{attribute 'linkalways'} 
{attribute 'no_explicit_call' := 'This FB is a CLASS and must be accessed using methods or properties'}
{attribute 'enable_dynamic_creation'}
FUNCTION_BLOCK _ETcVnTemplateMatchMethod EXTENDS EnumDatatypeBase
VAR
	localData : ETcVnTemplateMatchMethod;
	activeData : REFERENCE TO ETcVnTemplateMatchMethod;
	enumBaseDatatype : _DINT(localData);
END_VAR

METHOD PRIVATE AddLocalEnumeration
VAR_INPUT
	Enumeration : T_MAXSTRING;
	Value : ETcVnTemplateMatchMethod;
END_VAR
AddEnumeration(Enumeration, Value);
END_METHOD

PROPERTY PUBLIC Address : PVOID
GET
Address := ADR(activeData);
END_GET
END_PROPERTY

METHOD PUBLIC ClearReference
VAR_INPUT
END_VAR
activeData REF= localData;
SetBaseDatatypeReference();
END_METHOD

METHOD PUBLIC Clone : I_Datatype
VAR
    pClone : POINTER TO _ETcVnTemplateMatchMethod;
END_VAR
pClone := __NEW(_ETcVnTemplateMatchMethod(InitialValue := Value));
Clone := pClone^;
END_METHOD

METHOD FB_init : BOOL
VAR_INPUT
	bInitRetains : BOOL; // if TRUE, the retain variables are initialized (warm start / cold start)
	bInCopyCode : BOOL;  // if TRUE, the instance afterwards gets moved into the copy code (online change)
	InitialValue : ETcVnTemplateMatchMethod;
END_VAR
localData := InitialValue;
AddBaseDatatype(enumBaseDatatype);
ClearReference();

AddLocalEnumeration('TCVN_TMM_SQDIFF', ETcVnTemplateMatchMethod.TCVN_TMM_SQDIFF);
AddLocalEnumeration('TCVN_TMM_SQDIFF_NORMED', ETcVnTemplateMatchMethod.TCVN_TMM_SQDIFF_NORMED);
AddLocalEnumeration('TCVN_TMM_CCORR', ETcVnTemplateMatchMethod.TCVN_TMM_CCORR);
AddLocalEnumeration('TCVN_TMM_CCORR_NORMED', ETcVnTemplateMatchMethod.TCVN_TMM_CCORR_NORMED);
AddLocalEnumeration('TCVN_TMM_CCOEFF', ETcVnTemplateMatchMethod.TCVN_TMM_CCOEFF);
AddLocalEnumeration('TCVN_TMM_CCOEFF_NORMED', ETcVnTemplateMatchMethod.TCVN_TMM_CCOEFF_NORMED);
END_METHOD

PROPERTY PUBLIC Identifier : T_MAXSTRING
GET
Identifier := 'ETcVnTemplateMatchMethod';
END_GET
END_PROPERTY

METHOD IsEnumeratorValueEqual : BOOL
VAR_INPUT
	Enumerator : I_KeyValueForwardEnumerator;
END_VAR
VAR
	storedValue : ETcVnTemplateMatchMethod;
END_VAR
IF NOT Enumerator.TryGet(storedValue) THEN
	RETURN;
END_IF

IsEnumeratorValueEqual := storedValue = activeData;
END_METHOD

METHOD PUBLIC MakeReferenceTo
VAR_INPUT
	ReferenceTarget : REFERENCE TO ETcVnTemplateMatchMethod;
END_VAR
activeData REF= ReferenceTarget;
SetBaseDatatypeReference();
END_METHOD

METHOD PROTECTED SetBaseDatatypeReference
VAR_INPUT
END_VAR
enumBaseDatatype.MakeReferenceTo(activeData);
END_METHOD

PROPERTY PUBLIC Size : UDINT
GET
Size := SIZEOF(activeData);
END_GET
END_PROPERTY

METHOD TryMakeReferenceTo : BOOL
VAR_INPUT
	Target : I_Datatype;
END_VAR
VAR
	targetAsEnum : I_EnumDatatype;
	pTargetData : POINTER TO ETcVnTemplateMatchMethod;
END_VAR
IF NOT Target.TryResolveAsEnumDatatype(targetAsEnum) THEN
	RETURN;
END_IF

IF targetAsEnum.Identifier <> Identifier THEN
	RETURN;
END_IF

pTargetData := Target.Address;
activeData REF= pTargetData^;
SetBaseDatatypeReference();
TryMakeReferenceTo := TRUE;
END_METHOD

PROPERTY PUBLIC Value : ETcVnTemplateMatchMethod
GET
Value := activeData;
END_GET
SET
activeData := Value;
END_SET
END_PROPERTY

END_FUNCTION_BLOCK

(* stored: Version 1.1.0.1, ProductVersion 3.1.4024.12
   POU _ETcVnTemplateMatchMethod: Id {df4ea9b7-a56b-485e-a602-7928e7495125}, SpecialFunc None
   Folder Constructor: Id {6a73a42a-460b-4d52-ae9a-32c4e5d58b86}
   Folder Private: Id {29cd990b-ab22-4bc6-8de3-21ba69ec5868}
   Folder Protected: Id {6406afc1-ed90-4124-b098-a84d09e1c4b1}
   Method AddLocalEnumeration: Id {4bbc5cff-ba48-49df-ad14-3b1679e8d419}
   Property Address: Id {00671f9f-a90c-451a-9417-8433b6836364}
   Get Get: Id {e43d2360-eb3e-43e4-81fa-8ecf00ab023b}
   Method ClearReference: Id {fb3eda1a-dba8-41b3-b4d8-9b9372e0cd7e}
   Method Clone: Id {dc972ce0-6d43-4b17-99be-111b2fde3c56}
   Method FB_init: Id {28d73f06-2276-49dd-a9e4-744487b63a1e}
   Property Identifier: Id {e804da97-c467-44cd-8f5f-ddd76ab64e38}
   Get Get: Id {8cfa754d-a36e-4dbf-b1af-535facef67c1}
   Method IsEnumeratorValueEqual: Id {ca5b716e-f745-4017-97da-862ad4854a8a}
   Method MakeReferenceTo: Id {b21aca97-3aeb-486e-bb7f-c5002e9f63bc}
   Method SetBaseDatatypeReference: Id {d60542d6-10dc-4953-a31b-4992626f18f0}
   Property Size: Id {0db58dc0-db61-4ff4-96ad-4edbb021146b}
   Get Get: Id {77411c3c-eb4c-49f8-9b91-fd00389e45dd}
   Method TryMakeReferenceTo: Id {51bd588e-0a19-43c3-8461-dad2ba9a073d}
   Property Value: Id {efd2ba35-2f67-4d8e-b6d2-294e0e2b59f5}
   Get Get: Id {4834c36f-bc66-4696-bcf6-e7cc101289f4}
   Set Set: Id {2da8080a-2135-44b1-bf66-fda8dd99c388} *)
